{attribute 'qualified_only'}
VAR_GLOBAL
END_VAR

(* stored: Version 1.1.0.1, ProductVersion 3.1.4024.12
   GVL InputGVL_ControlBox: Id {0f4296d2-c735-406c-bb1d-db5f2a8b1826} *)
